{attribute 'qualified_only'}
{attribute 'strict'}
TYPE
E_BufferMode :
(
  Aborting := 0,
  Buffered := 1,
  BlendingJoint := 6,
  BlendingCartesian := 7
);
END_TYPE

(* stored: Version 1.1.0.1
   DUT E_BufferMode: Id {b5e72090-5cce-4c5c-a308-fa1602564a0a} *)
